FUNCTION_BLOCK TTestEventHandler IMPLEMENTS ITestEventHandler
VAR
    _EventWasRaised : BOOL;
    _EventData : UDINT;
END_VAR

PROPERTY EventWasRaised : BOOL
GET
EventWasRaised := _EventWasRaised;
END_GET
END_PROPERTY

METHOD OnCustomEvent
VAR_INPUT
    EventArgs : IStreamReader;
END_VAR
_EventData := EventArgs.Read_UDINT();
_EventWasRaised := TRUE;
END_METHOD

END_FUNCTION_BLOCK

(* stored: Version 1.1.0.1, ProductVersion 3.1.4024.4
   POU TTestEventHandler: Id {d6d2fc32-762c-41a8-95d4-a28d4a87bcac}, SpecialFunc None
   Property EventWasRaised: Id {53b0c48d-56ec-4d00-a4b8-81f80a9d2bac}
   Get Get: Id {1fe3e0fa-8dee-4a0c-969b-d371e197cc0f}
   Method OnCustomEvent: Id {982a11a9-f5f0-4911-b126-6808605ccf37} *)
